// TIA Portal project "R2D2" (V20)

(* hardware
DEVICE "R2D2"  S7-1200 Station
   slot 0: "Rack_0"  S7-1200 Rack  Rack  V1.0
   slot 1: "R2D2"  CPU 1212C DC/DC/DC  6ES7 212-1AE40-0XB0  V4.6
*)

// ===== PLC "R2D2"  CPU 1212C DC/DC/DC =====

TYPE "Crossroad_Input"
   STRUCT
      btnStart : Bool := FALSE;
      btnPause : Bool := FALSE;
      btnStop : Bool := FALSE;
      btnWestCrosswalk1 : Bool := FALSE;
      btnWestCrosswalk2 : Bool := FALSE;
      btnEastCrosswalk1 : Bool := FALSE;
      btnEastCrosswalk2 : Bool := FALSE;
      spare1 : DWord := 0;
      spare2 : DWord := 0;
      spare3 : DWord := 0;
      spare4 : DWord := 0;
   END_STRUCT;
END_TYPE

TYPE "Crossroad_Output"
   STRUCT
      crossroadType : Bool := FALSE;
      trafficLightNorth_green : Bool := FALSE;
      trafficLightNorth_yellow : Bool := FALSE;
      trafficLightNorth_red : Bool := FALSE;
      trafficLightSouth_green : Bool := FALSE;
      trafficLightSouth_yellow : Bool := FALSE;
      trafficLightSouth_red : Bool := FALSE;
      trafficLightWest_green : Bool := FALSE;
      trafficLightWest_yellow : Bool := FALSE;
      trafficLightWest_red : Bool := FALSE;
      trafficLightEast_green : Bool := FALSE;
      trafficLightEast_yellow : Bool := FALSE;
      trafficLightEast_red : Bool := FALSE;
      pedestrianSouth1_green : Bool := FALSE;
      pedestrianSouth1_red : Bool := FALSE;
      pedestrianSouth2_green : Bool := FALSE;
      pedestrianSouth2_red : Bool := FALSE;
      pedestrianWest1_green : Bool := FALSE;
      pedestrianWest1_red : Bool := FALSE;
      pedestrianWest2_green : Bool := FALSE;
      pedestrianWest2_red : Bool := FALSE;
      spare1 : DWord := 0;
      spare2 : DWord := 0;
      spare3 : DWord := 0;
      spare4 : DWord := 0;
   END_STRUCT;
END_TYPE

TYPE "Crosswalk_Input"
   STRUCT
      btnStart : Bool := FALSE;
      btnPause : Bool := FALSE;
      btnStop : Bool := FALSE;
      btnCrosswalk1 : Bool := FALSE;
      btnCrosswalk2 : Bool := FALSE;
      spare1 : DWord := 0;
      spare2 : DWord := 0;
      spare3 : DWord := 0;
      spare4 : DWord := 0;
   END_STRUCT;
END_TYPE

TYPE "Crosswalk_Output"
   STRUCT
      crosswalkType : Bool := FALSE;
      trafficLightGreen1 : Bool := FALSE;
      trafficLightsYellow1 : Bool := FALSE;
      trafficLightsRed1 : Bool := FALSE;
      trafficLightGreen2 : Bool := FALSE;
      trafficLightsYellow2 : Bool := FALSE;
      trafficLightsRed2 : Bool := FALSE;
      pedestrianLightGreen1 : Bool := FALSE;
      pedestrianLightRed1 : Bool := FALSE;
      pedestrianLightGreen2 : Bool := FALSE;
      pedestrianLightRed2 : Bool := FALSE;
      spare1 : DWord := 0;
      spare2 : DWord := 0;
      spare3 : DWord := 0;
      spare4 : DWord := 0;
   END_STRUCT;
END_TYPE

TYPE "Regulator_Input"
   STRUCT
      btnReset : Bool := FALSE;
      switchstate : Bool := FALSE;
      order : Int := 1;
      R1 : Real := 0.0;
      R2 : Real := 0.0;
      C1 : Real := 0.0;
      C2 : Real := 0.0;
      Uc1 : Real := 0.0;
      Uc2 : Real := 0.0;
      Td : Real := 0.0;
      Ts : Real := 0.0;
      spare1 : DWord := 0;
      spare2 : DWord := 0;
      spare3 : DWord := 0;
      spare4 : DWord := 0;
   END_STRUCT;
END_TYPE

TYPE "Regulator_Output"
   STRUCT
      Uin : Real := 0.0;
      spare1 : DWord := 0;
      spare2 : DWord := 0;
      spare3 : DWord := 0;
      spare4 : DWord := 0;
   END_STRUCT;
END_TYPE

TYPE "CarLight_Input"
   STRUCT
      btnReset : Bool := FALSE;
      error : Bool := FALSE;
      sensorLight : Bool := FALSE;
      sensorConnectorConnected : Bool := FALSE;
      lowBeamLight : Bool := FALSE;
      highBeamLight : Bool := FALSE;
      turnLight : Bool := FALSE;
      spare1 : DWord := 0;
      spare2 : DWord := 0;
      spare3 : DWord := 0;
      spare4 : DWord := 0;
   END_STRUCT;
END_TYPE

TYPE "CarLight_Output"
   STRUCT
      result : Bool := FALSE;
      spare1 : DWord := 0;
      spare2 : DWord := 0;
      spare3 : DWord := 0;
      spare4 : DWord := 0;
   END_STRUCT;
END_TYPE

DATA_BLOCK "DB_ProcessData"   // DB1
{ S7_Optimized_Access := 'FALSE' }
VERSION : 0.1
   VAR
      crossroad_input : "Crossroad_Input";
      crossroad_output : "Crossroad_Output";
      crosswalk_input : "Crosswalk_Input";
      crosswalk_output : "Crosswalk_Output";
      regulator_input : "Regulator_Input";
      regulator_output : "Regulator_Output";
      carlight_input : "CarLight_Input";
      carlight_output : "CarLight_Output";
   END_VAR
BEGIN
END_DATA_BLOCK

ORGANIZATION_BLOCK "Main"   // OB1, LAD, ProgramCycle
TITLE = "Main Program Sweep (Cycle)"
{ S7_Optimized_Access := 'TRUE' }
VERSION : 0.1
   VAR_INPUT
      Initial_Call : Bool;   // Initial call of this OB
      Remanence : Bool;   // =True, if remanent data are available
   END_VAR
BEGIN
END_ORGANIZATION_BLOCK